(* LS Electric XG5000 project: 241002_실습2 저수위 검출 *)
(* PLC LSPLC *)
(* module base 0 slot 0: 입력 모듈:XGI-D21A (DC 24V 입력, 8점 (전류소스/싱크입력)) *)
(* module base 0 slot 1: 출력 모듈:XGQ-RY1A (릴레이 출력, 8점 (2A용, 단독 COM.)) *)

PROGRAM NewProgram (* task: 스캔 프로그램 *)
VAR
    고수위 AT %IX0.0.0 : BOOL;
    저수위 AT %IX0.0.2 : BOOL;
    중수위 AT %IX0.0.1 : BOOL;
    펌프1 AT %QX0.1.0 : BOOL;
    펌프2 AT %QX0.1.1 : BOOL;
END_VAR

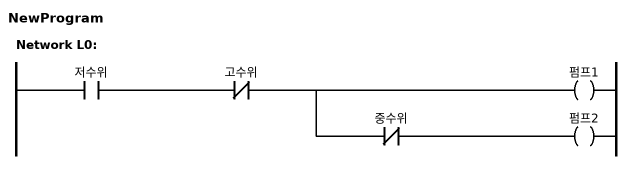
(* Rung L0 *)
펌프1 := 저수위 AND NOT 고수위;
펌프2 := 저수위 AND NOT 고수위 AND NOT 중수위;
END_PROGRAM